TYPE ST_HeightTest_CycleData :
STRUCT
	/////////////////////////////////////////////////////////////////////////////////////SETTINGS/////////////////////////////////////////////////////////////////////////////////////			
(**************************************************************************CURRENT SETTINGS DURING CYCLE. VELOCITY FOR EXAMPLE****************************************************)	
	
	anDistanceCalibrationBlock				: ARRAY [1..3] OF REAL;	
	anExpectedDistances						: ARRAY [1..3] OF REAL;	
	anHeightSetByCalibration				: ARRAY [1..4] OF REAL;	
	anTolerances							: ARRAY [1..3] OF REAL;	
	
	
/////////////////////////////////////////////////////////////////////////////////////GENERAL DATA/////////////////////////////////////////////////////////////////////////////////////			
(**************************************************************************RESULT DATA OF THE CYCLE. DISTANCE FOR EXAMPLE************************************************************)	
	
	anDistancesResult						: ARRAY [1..3] OF REAL;
	anRawMeasurement						: ARRAY [1..4] OF REAL; 

////////////////////////////////////////////////////////////////////////////////////RESULTS////////////////////////////////////////////////////////////////////////////////////////
(**************************************************************************DETERMINE IF THE PART FAIL OR PASS*********************************************************************)

	bPass				: BOOL;
	bFail				: BOOL;		

END_STRUCT
END_TYPE

(* stored: Version 1.1.0.1, ProductVersion 3.1.4026.17
   DUT ST_HeightTest_CycleData: Id {9fa01127-d8b3-4cd4-8460-18bade0da36e} *)
